{attribute addProperty BoxType "KL9900-0055"}
{attribute addProperty Id "Channel_1Channel_0AC2948E00"}
{attribute addProperty CRC "2573704743"}
{attribute addProperty SizeInBites "0"}
{attribute addProperty SizeInBytes "0"}
TYPE KL_99679E27 :
STRUCT
	{attribute addProperty Name "Channel_1"}
	Channel_1 : Channel_0AC2948E;
END_STRUCT
END_TYPE

(* stored: Version 1.2.0.0, ProductVersion 3.1.4024.9
   DUT KL_99679E27: Id {05b03df1-5266-4192-928d-b1329b8a215f} *)
